(* IEC 61131-3 sources: Lasal/CPU_5344_V01/Class/lampControlCurrentTwoZones, 1 file *)

(* ---- lampControlCurrentTwoZones.st ---- *)
(*!
<Class
	Name               = "lampControlCurrentTwoZones"
	Revision           = "0.0"
	RealtimeTask       = "false"
	CyclicTask         = "true"
	DefCyclictime      = "10 ms"
	BackgroundTask     = "false"
	Sigmatek           = "false"
	OSInterface        = "false"
	HighPriority       = "false"
	Automatic          = "false"
	UpdateMode         = "Prescan"
	SharedCommandTable = "true"
	Objectsize         = "(420,300)">
	<Channels>
		<Server Name="ClassSvr" Visualized="false" Initialize="false" WriteProtected="true" Retentive="false"/>
		<Server Name="zone2" Visualized="false" Initialize="true" DefValue="1" WriteProtected="false" Retentive="false"/>
		<Server Name="zone3" Visualized="false" Initialize="true" DefValue="1" WriteProtected="false" Retentive="false"/>
		<Server Name="zoneMain" Visualized="false" Initialize="false" WriteProtected="false" Retentive="false"/>
		<Client Name="iBlinkMain" Required="true" Internal="false"/>
		<Client Name="iBlinkZone2" Required="true" Internal="false"/>
		<Client Name="oLight" Required="true" Internal="false"/>
	</Channels>
</Class>
*)
lampControlCurrentTwoZones : CLASS
  //Servers:
	ClassSvr 	: SvrChCmd_DINT;
	zoneMain 	: SvrCh_DINT;
	zone2 	: SvrCh_DINT;
	zone3 	: SvrCh_DINT;
  //Clients:
	iBlinkMain 	: CltCh_DINT;
	iBlinkZone2 	: CltCh_DINT;
	oLight 	: CltCh_DINT;
  //Variables:
  //Functions:

	FUNCTION VIRTUAL GLOBAL CyWork
		VAR_INPUT
			EAX 	: UDINT;
		END_VAR
		VAR_OUTPUT
			state (EAX) 	: UDINT := READY;
		END_VAR;
  //Tables:
	FUNCTION @STD
		VAR_OUTPUT
			ret_code	: CONFSTATES;
		END_VAR;
	FUNCTION GLOBAL TAB @CT_;
END_CLASS;

// JdK 14-10-2020 lampControlCurrentTwoZones, goal is to let lamp blink if one of the zones is in blink mode, else just on or off

FUNCTION VIRTUAL GLOBAL lampControlCurrentTwoZones::CyWork
	VAR_INPUT
		EAX 	: UDINT;
	END_VAR
	VAR_OUTPUT
		state (EAX) 	: UDINT;(* := READY *)
	END_VAR

  iBlinkMain:= iBlinkMain.Read();
  iBlinkZone2:= iBlinkZone2.Read();

  IF zoneMain= 1 THEN
    IF zone2= 0 | zone3= 0 THEN
      oLight:= 0;
    ELSIF zone2= 2 | zone3=2 THEN
      oLight:= iBlinkZone2;
    ELSE
      oLight:= 1;
    END_IF;
  ELSIF zoneMain= 2 & zone2>= 1 & zone3>= 1 THEN
    oLight:= iBlinkMain;
  ELSE
    oLight:= 0;
  END_IF;

  oLight.Write(input:=oLight);

END_FUNCTION
